{attribute 'OPC.UA.DA.StructuredType' := '1'}
TYPE MessageDescription :
STRUCT
	Severity: eSeverity;				//Info, Warning, Error, Critical
	Category: eMessageCategories;	//MissingInfo, NotImplemented etc.
	sSender: STRING;				//Beschreibung von User z.B. FB_Befüllen
	sMessage: STRING;				//Beschreibung von User z.B. "Tank bereits voll"
	tTime: TIME;					//Zeitpunkt wann Message generiert wurde
	bQuit: BOOL;					//Message wurde von User quittiert
	ID: UINT;						//ID von Message
	
END_STRUCT
END_TYPE

(* stored: Version 1.1.0.1, ProductVersion 3.1.4026.18
   DUT MessageDescription: Id {39ffd807-d9e4-4c8b-9d95-0d96aa3e820a} *)
